PROGRAM POU_AxisJogCtrl
VAR
	fb_Axis1Jog: MC_Jog;
	fb_Axis2Jog: MC_Jog;
END_VAR

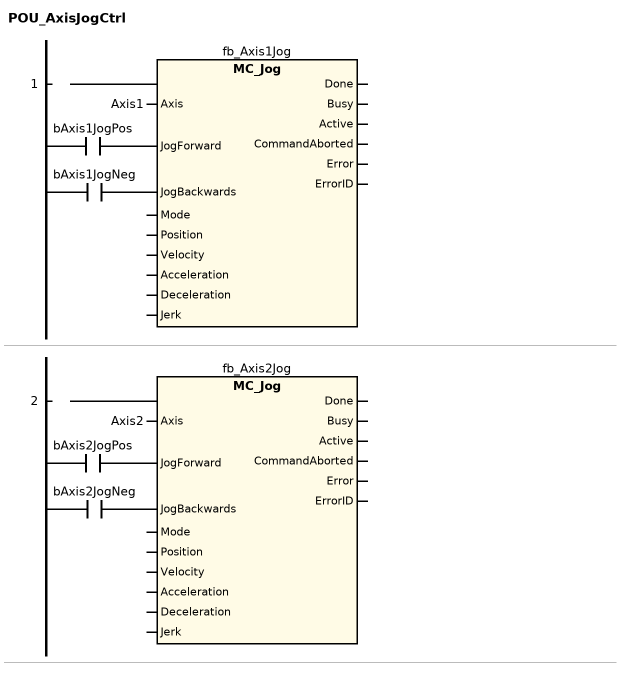
// NETWORK 1
fb_Axis1Jog(Axis := Axis1, JogForward := bAxis1JogPos, JogBackwards := bAxis1JogNeg); // MC_Jog

// NETWORK 2
fb_Axis2Jog(Axis := Axis2, JogForward := bAxis2JogPos, JogBackwards := bAxis2JogNeg); // MC_Jog

END_PROGRAM

(* stored: Version 1.1.0.1, ProductVersion 3.1.4022.18
   POU POU_AxisJogCtrl: Id {6be64ff8-130d-4b4b-ad49-9160c0c676c9}, SpecialFunc None *)
